VAR_GLOBAL
	bool_value : bool;
END_VAR

(* stored: Version 1.1.0.1, ProductVersion 3.1.4024.0
   GVL global: Id {f3f9bbc8-0bb6-435c-9a30-6bff361b4fb3} *)
